FUNCTION_BLOCK TrajectoryController IMPLEMENTS  TrajectoryControllable
VAR_INPUT
	//Freigabesignal für Fahrt, Roboter stoppt bei FALSE
	xBoEnable: 					BOOL := FALSE;
	
	//Anfahrt (in Sperrzone vor Tasche oder Ladestation) = 1, Fahrt = 0
	xIntMoveToEndPosition: INT := 0;
END_VAR
VAR_OUTPUT
	//TRUE, wenn Ziel erreicht, Ziel entspricht letzten gültigen WP
	yBoArrivedAtDestination: 	BOOL := FALSE;
	
	//TRUE, wenn der Roboter fährt
	yBoDriving: 				BOOL := FALSE;
	
	//COUNTER zur Anzeige, des Indexes des nächstes WP
	yUintWaypointIndex: 		BOOL := 0;
	
	//aktuelle Roboterposition, für Simulationszwecke
	yRPposition: 				RobotPose;
	
END_VAR
VAR
END_VAR

{warning 'Eigenschaftenimplementierung hinzufügen'}
PROPERTY ArrivedAtDestination : BOOL
GET
END_GET
SET
END_SET
END_PROPERTY

{warning 'Eigenschaftenimplementierung hinzufügen'}
PROPERTY Driving : BOOL
GET
END_GET
SET
END_SET
END_PROPERTY

{warning 'Eigenschaftenimplementierung hinzufügen'}
PROPERTY Enable : BOOL
GET
END_GET
SET
END_SET
END_PROPERTY

{warning 'Eigenschaftenimplementierung hinzufügen'}
PROPERTY RobotPose : RobotPose
GET
END_GET
SET
END_SET
END_PROPERTY

{warning 'Methodenimplementierung hinzufügen'}
METHOD setWaypointList
VAR_INPUT
	WaypointList	: ARRAY [1...30] OF RobotPose;
END_VAR
END_METHOD

{warning 'Eigenschaftenimplementierung hinzufügen'}
PROPERTY WaypointIndex : UINT
GET
END_GET
SET
END_SET
END_PROPERTY

{warning 'Eigenschaftenimplementierung hinzufügen'}
(*TODO: define max number of waypoints!*)
PROPERTY WaypointList : ARRAY [1...!!!'ERROR'!!!] OF RobotPose
GET
END_GET
SET
END_SET
END_PROPERTY

END_FUNCTION_BLOCK

(* stored: Version 1.1.0.1, ProductVersion 3.1.4024.11
   POU TrajectoryController: Id {8d8b1656-17ec-4ef2-9a7c-c3047fa0f4d8}, SpecialFunc None
   Property ArrivedAtDestination: Id {8c53fe4c-633d-475e-8a27-006b1a2fd284}
   Get Get: Id {deaf1f9b-6394-410e-a97f-5698a8ab83ec}
   Set Set: Id {561fbf8b-a0cd-474b-b582-ac0e45e0d919}
   Property Driving: Id {0905c582-29a2-452f-a9ba-c41fbe353ae5}
   Get Get: Id {8451708f-658e-4458-836e-518765e2f5d8}
   Set Set: Id {7482c7e8-2785-48cc-be2f-5ab1da2da63a}
   Property Enable: Id {6e573747-6921-4d90-932b-ae7342a97885}
   Get Get: Id {b28a8887-cce3-46bc-b1bd-f4d08148a174}
   Set Set: Id {90f6f9db-6f2a-43c5-9ff0-786fbaa1d944}
   Property RobotPose: Id {5458479b-1905-4ad8-915e-7c40700f6181}
   Get Get: Id {9482d3aa-f011-4fb8-873a-7e15ede74c4b}
   Set Set: Id {1f5e8a03-b842-44a4-a300-f8f33ff2fb86}
   Method setWaypointList: Id {a5914345-393a-4c37-a337-155a4553329f}
   Property WaypointIndex: Id {0b02d2b3-24cb-45b9-bc2d-73a80c8e7123}
   Get Get: Id {1a404b8c-d0e0-4cb3-b9a9-964d8b21427b}
   Set Set: Id {0b680c3e-8f7e-4f48-872a-644443530364}
   Property WaypointList: Id {31729257-f6ad-4e64-b69d-baa1e11be102}
   Get Get: Id {c07493c7-6255-4ec1-9fbe-73733b144694}
   Set Set: Id {8f5b2748-2097-49f7-ad4f-d3d53075efa5} *)
